FUNCTION_BLOCK FB_Component_Indicator EXTENDS FB_ComponentBase_SR IMPLEMENTS I_Indicator
VAR

    // Outputs

    IndicatorOutput AT %Q* : BOOL;

    // HMI

    Indicator_HMI : ST_Indicator_HMI;

    // Alarms

    IndicatorAlarms : ARRAY[1..Indicator_ALARMS_COUNT] OF FB_TcAlarm;

    // Internal variables

    Pulse     : FB_PulseGenerator;
    _Flashing : BOOL;
    _On       : BOOL;

END_VAR

VAR CONSTANT
    Indicator_ALARMS_COUNT : UDINT := 5;
END_VAR

METHOD PROTECTED CreateEvents
VAR_INPUT
END_VAR
F_CreateAllEventsInClass(Alarms     := IndicatorAlarms,
                         ClassSize  := SIZEOF(TC_EVENTS.ComponentBase),
                         pInitEvent := ADR(TC_EVENTS.ComponentBase.InitReferenceEvent),
                         Prefix     := _Name);

SUPER^.CreateEvents();
END_METHOD

//! @summary This method serves as the entry point for all underlying FB logic
METHOD PUBLIC CyclicLogic

//! @description This method should be called cyclically by descendant function blocks by invoking <c>SUPER^.CyclicLogic()</c>.  Alternatively, the contents of this method could be reimplemented entirely in which case a call to this method would not be necessary.
// Initialise Component

IF NOT _InitComplete THEN
    _InitComplete := Initialize();
    RETURN;
END_IF

IF _Flashing THEN
    Pulse.CyclicLogic();
    IndicatorOutput := Pulse.PulseOutput;
END_IF

// Call Super

SUPER^.CyclicLogic();

// Set Current Alarm Severity

_CurrentAlarmSeverity := F_GetMaxSeverityRaised(Alarms := IndicatorAlarms, CurrentSeverity := _CurrentAlarmSeverity);
END_METHOD

METHOD Flash
_Flashing := TRUE;
_On       := FALSE;

IndicatorOutput := Pulse.PulseOutput;
END_METHOD

PROPERTY Flashing : BOOL
GET
Flashing := _Flashing;
END_GET
END_PROPERTY

//! @summary Basic component initialization logic
METHOD PROTECTED Initialize : BOOL;

//! @description This method is called by <c>CyclicLogic()</c> as required
CreateEvents();

IF SUPER^.Initialize() THEN
    Initialize := TRUE;
END_IF
END_METHOD

METHOD PROTECTED Monitoring
VAR_INPUT
END_VAR
IF NOT IndicatorAlarms[E_ComponentBase.SimulationWarning].bRaised AND _Simulate AND NOT Parameters_BaseComponent.INHIBIT_SIMULATION_WARNING THEN
    IndicatorAlarms[E_ComponentBase.SimulationWarning].Raise(0);
ELSIF IndicatorAlarms[E_ComponentBase.SimulationWarning].bRaised AND NOT _Simulate THEN
    IndicatorAlarms[E_ComponentBase.SimulationWarning].Clear(0, 0);
END_IF

_CurrentAlarmSeverity := TcEventSeverity.Verbose;
_CurrentAlarmSeverity := F_GetMaxSeverityRaised(Alarms := IndicatorAlarms, CurrentSeverity := _CurrentAlarmSeverity);

SUPER^.Monitoring();
END_METHOD

PROPERTY Off : BOOL
GET
Off := NOT _ON AND NOT _Flashing;
END_GET
END_PROPERTY

PROPERTY PUBLIC OffTime : TIME
SET
Pulse.OffTime := OffTime;
END_SET
END_PROPERTY

PROPERTY On : BOOL
GET
On := _On;
END_GET
END_PROPERTY

PROPERTY PUBLIC OnTime : TIME
SET
Pulse.OnTime := OnTime;
END_SET
END_PROPERTY

METHOD Reset : BOOL
TurnOff();
END_METHOD

METHOD TurnOff
_Flashing := FALSE;
_On       := FALSE;

IndicatorOutput := FALSE;
END_METHOD

METHOD TurnOn
_Flashing := FALSE;
_On       := TRUE;

IndicatorOutput := TRUE;
END_METHOD

END_FUNCTION_BLOCK

(* stored: Version 1.1.0.1
   POU FB_Component_Indicator: Id {ed010e85-f1ac-4322-94b7-f14d6f0299c2}, SpecialFunc None
   Folder I_ComponentBase: Id {793a438e-8b4a-4273-ae98-184afab389a8}
   Folder I_CyclicFB: Id {50934f65-5f9a-44db-97b1-1e0e0dc03e17}
   Folder I_Template: Id {e5565f98-12ce-47de-8158-4b402d784447}
   Folder Methods: Id {fded1359-9773-4033-b1fe-88cbfb8a401d}
   Folder Properties: Id {8661cad9-cc95-43a0-b387-4594bd6b4ed5}
   Method CreateEvents: Id {69edbd4a-9cc7-4356-bdca-17f708619a85}
   Method CyclicLogic: Id {7d2b89bf-8791-4bb0-8e73-3f76c01a9fec}
   Method Flash: Id {f458df86-8ff5-4edd-9fa2-e0993ba9901f}
   Property Flashing: Id {a4932e8a-4897-42c7-9759-38925d2788f1}
   Get Get: Id {ac1ef52a-ab08-49a2-acec-3bf1ef59baed}
   Method Initialize: Id {0c76f14f-9965-435e-b292-3902454f980e}
   Method Monitoring: Id {7f222f43-eff7-4b11-8b5c-f0394503bee1}
   Property Off: Id {30d8980a-b740-4677-91ca-eac87f3a7208}
   Get Get: Id {c5c4328e-ab5e-4ee2-aa53-6d1ad7cadadf}
   Property OffTime: Id {c57b4239-6948-4ad9-bedf-672d8178212a}
   Set Set: Id {dc6c845c-63d2-494b-819c-ede682509e15}
   Property On: Id {7fc3cb81-daf4-4bf2-84ed-048fafd66410}
   Get Get: Id {0e3a66aa-d69a-4ecb-9188-342af31e82d5}
   Property OnTime: Id {c847daa9-67e4-4b0a-bb54-7236e93d6c42}
   Set Set: Id {f0ab1366-ed32-4b5a-ba41-f8d23e416810}
   Method Reset: Id {330f7997-cdc7-4e1d-88f4-7a5a4af27f6a}
   Method TurnOff: Id {ab47395d-7219-4b5f-adac-e7e6852c78d9}
   Method TurnOn: Id {1ba73b21-cf21-4808-a6e0-c3003a413f0e} *)
